PROGRAM MAIN
VAR
	
MyMover : XplanarMover; 

MyController : XboxController; 

MyEnvironment : Environment; 

END_VAR

Cyclic(); 


MyMover(
	
MoverType := 'AMP4220'

); 


MyEnvironment.Boundry(

NumberOfXTiles := 4, 
NumberOfYTiles := 4	,
MoverTypeWidth 				:= MyMover.TypeWidth, 
MoverTypeLength				:= MyMover.TypeLength 
);

ACTION Cyclic:
//Initizalization
MyMover.Init( 
bStart := MyController.Start
);

//Recover 
MyMover.Recover(
bBack := MyController.Reset
); 

//tilt
MyMover.Tilt_Height(
rStick_X := MyController.rStick_X,
rStick_Y := MyController.rStick_Y,
bButton_B := MyController.Button_B,
LBumper := MyController.lBumper,
RBumper	:= MyController.rBumper
);

//X and Y Movement 
MyMover.XYMovement(
lStick_X := MyController.lStick_X, 
lStick_Y := MyController.lStick_Y, 
bButton_A := MyController.Button_A, 
bButton_X := MyController.Button_X, 
bButton_Y := MyController.Button_Y, 
maxXTravel := MyEnvironment.MaxTableXTravel,
minXTravel := MyEnvironment.MinTableXTravel,
maxYTravel := MyEnvironment.MaxTableYTravel,
minYTravel := MyEnvironment.MinTableYTravel,
);

MyMover.Rotation(
LTrigger := MyController.lTrigger,
RTrigger := MyController.rTrigger
);

MyController.takeScreenshot(
bDpad_D := Mycontroller.Dpad_D,
MoverPosition := MyMover.Xplanar_Mover.MCTOPLC.ACT.ActPos
);

MyController.clearScreenshot(
bDpad_U := MyController.Dpad_U,
ClearPosition := MyController.ZeroVector
);

MyMover(); 
MyController();
MyEnvironment();
END_ACTION

END_PROGRAM

(* stored: Version 1.1.0.1, ProductVersion 3.1.4024.12
   POU MAIN: Id {961e48bf-3b1b-48fd-8912-207c5805ebf3}, SpecialFunc None
   Action Cyclic: Id {b613598b-d147-44e5-bf73-b51c64ea6006} *)
